PROGRAM POU_Seguridad
VAR
	Emergency_Stop : BOOL := FALSE; // variable para indicar la parada inmediata de la planta
END_VAR

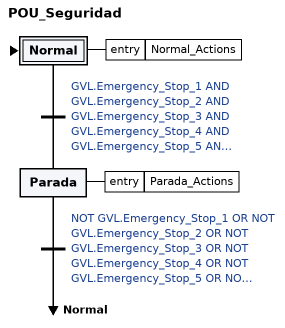
INITIAL_STEP Normal:
    Normal_Actions(P1);  // entry action
END_STEP
TRANSITION FROM Normal TO Parada
    := GVL.Emergency_Stop_1 AND GVL.Emergency_Stop_2 AND GVL.Emergency_Stop_3 AND GVL.Emergency_Stop_4 AND GVL.Emergency_Stop_5 AND GVL.Emergency_Stop_6 AND GVL.Emergency_Stop_7 AND GVL.Emergency_Stop_8 AND GVL.Emergency_Stop_9;
END_TRANSITION
STEP Parada:
    Parada_Actions(P1);  // entry action
END_STEP
TRANSITION FROM Parada TO Normal
    := NOT GVL.Emergency_Stop_1 OR NOT GVL.Emergency_Stop_2 OR NOT GVL.Emergency_Stop_3 OR NOT GVL.Emergency_Stop_4 OR NOT GVL.Emergency_Stop_5 OR NOT GVL.Emergency_Stop_6 OR NOT GVL.Emergency_Stop_7 OR NOT GVL.Emergency_Stop_8 OR NOT GVL.Emergency_Stop_9;
END_TRANSITION

ACTION Normal_Actions:
 Emergency_Stop := FALSE;
 //Se desactivan las alarmas
GVL.Alarm_Siren  := FALSE;
GVL.Warning_Light  := FALSE;
GVL.Factory_IO_Pause := FALSE;
END_ACTION

ACTION Parada_Actions:
 Emergency_Stop := TRUE;
 // Se indica mediante una luz que el siguiente botón a pulsar sería el de Reset
GVL.Stop_Button_2_Light := FALSE;
GVL.Reset_Button_2_Light := TRUE;
//Se activan las alarmas
GVL.Alarm_Siren  := TRUE;
GVL.Warning_Light  := TRUE;
POU_Parada();
END_ACTION

END_PROGRAM

(* stored: Version 1.1.0.1, ProductVersion 3.1.4024.12
   POU POU_Seguridad: Id {d6523909-5f41-498b-8353-e6c137019c24}, SpecialFunc None
   Action Normal_Actions: Id {ddcdd99b-0135-45e0-874d-763b32f62815}
   Action Parada_Actions: Id {3f4b4dce-d39a-4723-822b-8715087ef13c} *)
